PROGRAM PLC_PRG
VAR
	//Visualization Buttons
	mxButtonReset: BOOL;	
	mxButtonStart: BOOL;
	
	//Internal use
	mxComBusy: BOOL;
	mxStart: BOOL;	
	mxDone: BOOL;
	ComData: CommunicationData;
	
	//Motion Function Blocks
	fbCommunicator: Communicator;
	fbABBGoToHome_1: ABBGoToHome;
	fbABBGoToSensor_1: ABBGoToSensor;
	fbABBPickLeaveSensor_1: ABBPickLeaveSensor;
END_VAR

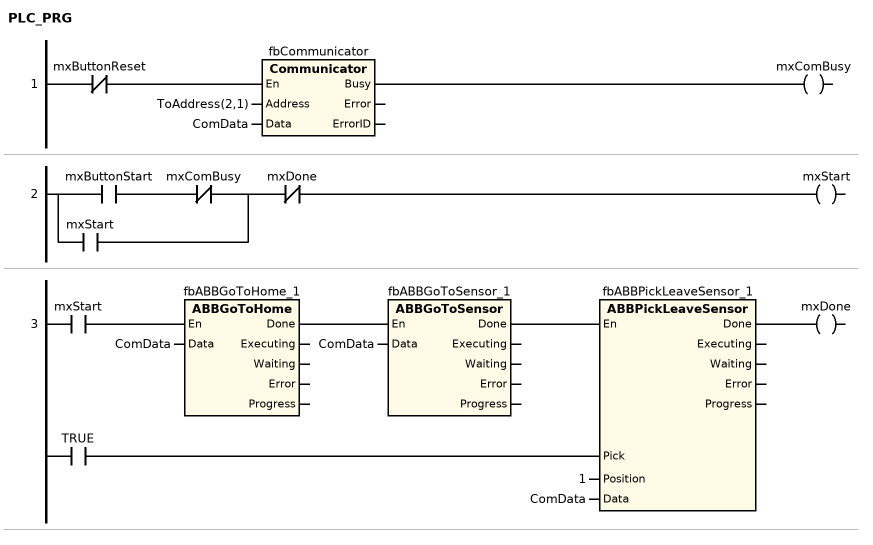
// NETWORK 1
fbCommunicator(En := NOT mxButtonReset, Address := ToAddress(2,1), Data := ComData); // Communicator
mxComBusy := fbCommunicator.Busy;

// NETWORK 2
mxStart := (mxButtonStart AND NOT mxComBusy OR mxStart) AND NOT mxDone;

// NETWORK 3
fbABBGoToHome_1(En := mxStart, Data := ComData); // ABBGoToHome
fbABBGoToSensor_1(En := fbABBGoToHome_1.Done, Data := ComData); // ABBGoToSensor
fbABBPickLeaveSensor_1(En := fbABBGoToSensor_1.Done, Pick := TRUE, Position := 1, Data := ComData); // ABBPickLeaveSensor
mxDone := fbABBPickLeaveSensor_1.Done;

END_PROGRAM

(* stored: Version 1.1.0.1, ProductVersion 3.1.4022.12
   POU PLC_PRG: Id {2ef04e23-149a-4400-a32c-9834775884e9}, SpecialFunc None *)
